Staubli VAL3: get.pgx

public program get(string& x_sItem[], num x_nIndex)
begin
end
